FUNCTION_BLOCK FB_Observable_LINT EXTENDS FB_AbstractObservable
VAR
    _nVal:              LINT;
    _nOldVal:           LINT;
END_VAR

METHOD FB_init : BOOL
VAR_INPUT
    bInitRetains:       BOOL; // if TRUE, the retain variables are initialized (warm start / cold start)
    bInCopyCode:        BOOL;  // if TRUE, the instance afterwards gets moved into the copy code (online change)
END_VAR
THIS^._nTypeClass := __SYSTEM.TYPE_CLASS.TYPE_LINT;
END_METHOD

PROPERTY nDataSize : UDINT
GET
nDataSize := SIZEOF(LINT);
END_GET
END_PROPERTY

PROPERTY nValue64 : LINT
GET
nValue64 := THIS^._nVal;
END_GET
SET
THIS^._nOldVal := THIS^._nVal;
THIS^._nVal := nValue64;

THIS^.NotifyWithConditions();
END_SET
END_PROPERTY

PROPERTY PROTECTED pData : POINTER TO BYTE
GET
pData := ADR(THIS^._nVal);
END_GET
END_PROPERTY

METHOD  ValueChanged : BOOL
VAR_INPUT
END_VAR
ValueChanged := THIS^._nOldVal <> THIS^._nVal;
END_METHOD

END_FUNCTION_BLOCK

(* stored: Version 1.1.0.1, ProductVersion 3.1.4024.12
   POU FB_Observable_LINT: Id {4f53a217-a7ed-07e9-3a6c-add2f2d343ab}, SpecialFunc None
   Method FB_init: Id {523d5c68-6c5e-0005-2ef6-4831c55b1d6d}
   Property nDataSize: Id {73aa52e9-7fe3-039f-3466-47276395b5e5}
   Get Get: Id {7a18b90b-a3b9-068a-1179-74ea9c32ca06}
   Property nValue64: Id {d250bcb8-857b-043c-3632-c0eb17f08ea9}
   Get Get: Id {324fb308-1178-027b-3048-030303ff1fc5}
   Set Set: Id {466d7844-01fd-0d76-212d-f891b5ca48ce}
   Property pData: Id {ad9d8f4a-b75b-0bde-14ee-f1f7d33437c0}
   Get Get: Id {f2bce764-acdb-0d9b-1f6d-553b09302ac1}
   Method ValueChanged: Id {b8f94696-391d-0d6f-293a-ff7203ea0756} *)
